Staubli VAL3: getLanguage.pgx

public program getLanguage(string& x_sPath[])
begin
  x_sPath=language:libPath()
end
